// Mitsubishi GX Works2 project: 수위문제   PLC: Q02/Q02H

PROGRAM MAIN
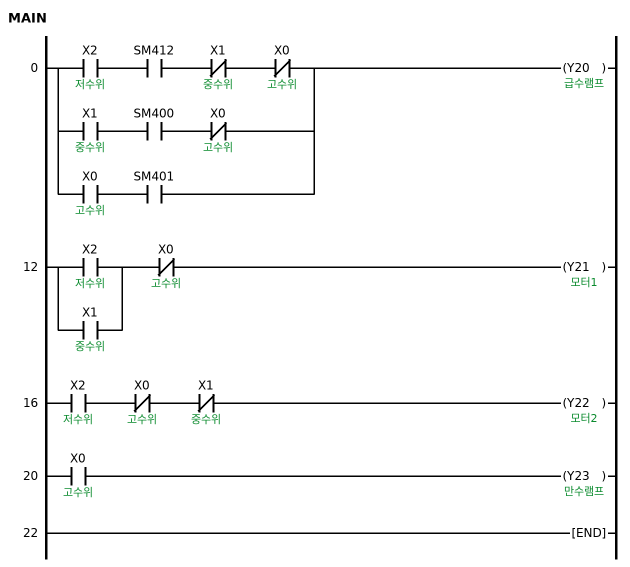
0     LD      X2  ; 저수위
      AND     SM412
      ANI     X1  ; 중수위
      ANI     X0  ; 고수위
      LD      X1  ; 중수위
      AND     SM400
      ANI     X0  ; 고수위
      ORB
      LD      X0  ; 고수위
      AND     SM401
      ORB
      OUT     Y20  ; 급수램프
12    LD      X2  ; 저수위
      OR      X1  ; 중수위
      ANI     X0  ; 고수위
      OUT     Y21  ; 모터1
16    LD      X2  ; 저수위
      ANI     X0  ; 고수위
      ANI     X1  ; 중수위
      OUT     Y22  ; 모터2
20    LD      X0  ; 고수위
      OUT     Y23  ; 만수램프
22    END
END_PROGRAM

// device comments not shown above
M0  ; 보조0
M1  ; 보조1
M2  ; 보조2
M3  ; 보조3
